FUNCTION_BLOCK FB_AXIS_CONTROL
VAR_IN_OUT
	IQAxisRef:					AXIS_REF;
END_VAR
VAR_INPUT
	IJogForward:				BOOL;
	IJogBackward:				BOOL;
	IStartPos: 					BOOL;
	ITargetPos:					LREAL;
	IJogMode:					E_JogMode;
	IPowerOn:					BOOL;
	IAckDone:					BOOL;
	IStepSize:					LREAL;
	IOverride:					LREAL;
	IManualOverride:			LREAL;
	IMaxVelocity:				LREAL;
END_VAR
VAR_OUTPUT
	QAxisReady:					BOOL;
	QActPos:					LREAL;
	QAxisDone:					BOOL;
END_VAR
VAR
	MCPower: 					MC_Power;
	toPowerOn: 					TON;
	MCMoveAbs_01: 				MC_MoveAbsolute;
	MCMoveAbs_02:				MC_MoveAbsolute;
	MCJog: 						MC_Jog;
	MCHalt: 					MC_Halt;
	MCReset: 					MC_Reset;
	SoEReset: 					FB_SoEReset;
	
	ErrorID:					UDINT;
	chNetId: 					STRING(23) := '';	
	lrTargetOldPos:				LREAL;
	lrManualOverride:			LREAL;
	xAxisDone:					BOOL;
	rtAxisDone:					R_TRIG;
	xSoeExecute:				BOOL;
	xTogglePos:					BOOL;
	xHalt:						BOOL;
	fbRefactor: REFACTOR_LREAL;
END_VAR
VAR // added by the converter: edge detectors and wires of the graphical bodies
    _w1 : BOOL;
END_VAR

(*Axis done on rise edge of xAxisDone bit and reset on external IAckDone*)
rtAxisDone(CLK:=(MCMoveAbs_01.Done OR MCMoveAbs_02.Done));

IF rtAxisDone.Q THEN
	QAxisDone:= TRUE;
	
ELSIF IAckDone AND QAxisDone THEN
	QAxisDone:= FALSE;
	lrTargetOldPos:=ITargetPos;
END_IF

(*Refactoring the speed for manual jogging*)
fbRefactor(	I_Percentage:= IManualOverride, 
			I_MaximumValue:= IMaxVelocity, 
			Q_Result=> lrManualOverride);

(*SoEReset execution on errors or if axis is not ready*)
xSoeExecute:= MCPower.Error OR MCMoveAbs_02.Error OR MCMoveAbs_01.Error OR MCJog.Error OR MCHalt.Error OR NOT QAxisReady;



(*T#300MS delay on PowerON*)
toPowerOn(IN:= IPowerOn, PT:= T#300MS);

(*Read axis actual position*)
QActPos:= IQAxisRef.NcToPlc.ActPos;

(*Trigger new target position*)
IF(lrTargetOldPos <> ITargetPos) THEN
	xTogglePos:= TRUE;
ELSE
	xTogglePos:= FALSE;
END_IF

xHalt:=(NOT IJogForward AND NOT IJogBackward) AND NOT MCHalt.Done;

MC_MOVE_ACT();

ACTION MC_MOVE_ACT:
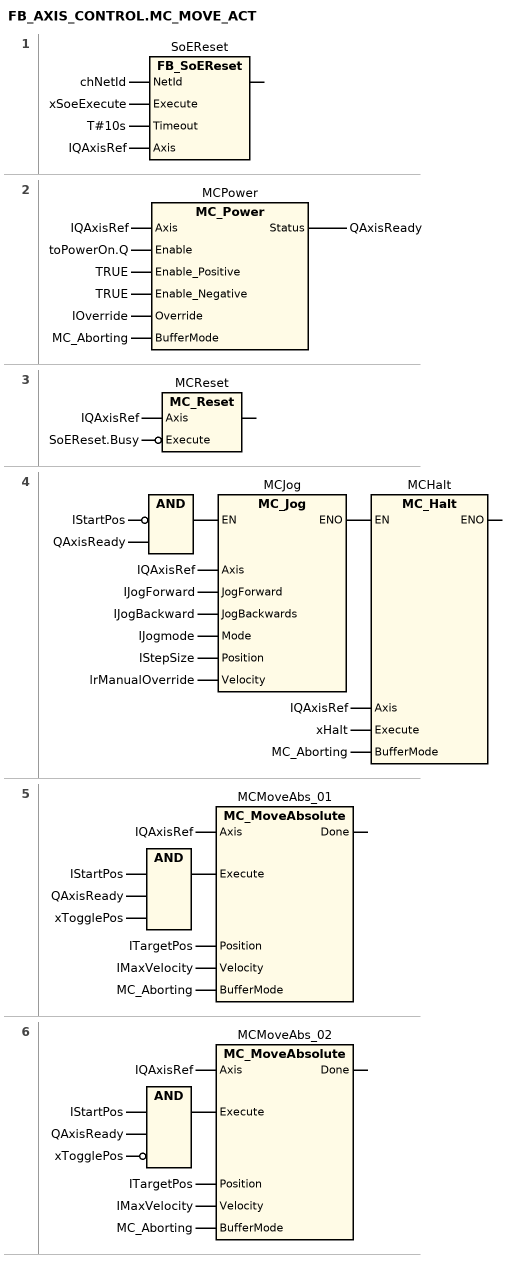
// NETWORK 1
SoEReset(NetId := chNetId, Execute := xSoeExecute, Timeout := T#10s, Axis := IQAxisRef); // FB_SoEReset

// NETWORK 2
MCPower(
    Axis := IQAxisRef,
    Enable := toPowerOn.Q,
    Enable_Positive := TRUE,
    Enable_Negative := TRUE,
    Override := IOverride,
    BufferMode := MC_Aborting); // MC_Power
QAxisReady := MCPower.Status;

// NETWORK 3
MCReset(Axis := IQAxisRef, Execute := NOT SoEReset.Busy); // MC_Reset

// NETWORK 4
_w1 := NOT IStartPos AND QAxisReady;
IF _w1 THEN
    MCJog(
        Axis := IQAxisRef,
        JogForward := IJogForward,
        JogBackwards := IJogBackward,
        Mode := IJogmode,
        Position := IStepSize,
        Velocity := lrManualOverride); // MC_Jog
END_IF
IF _w1 THEN
    MCHalt(Axis := IQAxisRef, Execute := xHalt, BufferMode := MC_Aborting); // MC_Halt
END_IF

// NETWORK 5
MCMoveAbs_01(
    Axis := IQAxisRef,
    Execute := IStartPos AND QAxisReady AND xTogglePos,
    Position := ITargetPos,
    Velocity := IMaxVelocity,
    BufferMode := MC_Aborting); // MC_MoveAbsolute

// NETWORK 6
MCMoveAbs_02(
    Axis := IQAxisRef,
    Execute := IStartPos AND QAxisReady AND NOT xTogglePos,
    Position := ITargetPos,
    Velocity := IMaxVelocity,
    BufferMode := MC_Aborting); // MC_MoveAbsolute
END_ACTION

END_FUNCTION_BLOCK

(* stored: Version 1.1.0.1, ProductVersion 3.1.4022.18
   POU FB_AXIS_CONTROL: Id {8fecf8b5-8ea7-4a09-9ff7-bab4f36a3cce}, SpecialFunc None
   Action MC_MOVE_ACT: Id {96dd3873-5cb0-4d2a-9390-6553a8cefe70} *)
